(* CODESYS project FU_iBitPartThrough.xml

Project tree, tasks and I/O mapping:
  function FU_iBitPartThrough [ST]
*)

// FU_iBitPartThrough
//This function changed only the needed bits of a variable
// |**Version**|**Author**| **Date** |**Changes**
// | 1         | NSN      | 16-03-22 | Creation
FUNCTION FU_iBitPartThrough : INT
VAR_INPUT
	valueChange		:INT;		//Variable to change
	value			:INT;		//Value to change bits to
	amount			:BYTE;		//Amount of bits to change
	offset			:BYTE;		//Offset in variable to change bits at
END_VAR

FU_iBitPartThrough		:=		TO_INT((TO_UINT(valueChange) AND ROL(TO_UINT(GConstants.binaryInvMaskInt[amount]),offset)) OR SHL(TO_UINT(value) AND TO_UINT(GConstants.binaryMaskInt[amount]),offset));

END_FUNCTION
